// TIA Portal V17 export
// export: Created 2025-06-25T13:13:16.5727411Z, ExportSetting WithDefaults, DisplayName Totally Integrated Automation Portal, DisplayVersion V17 Update 8, DisplayName TIA Portal Openness, DisplayVersion V17 Update 8, DisplayName TIA Portal Version Control Interface, DisplayVersion V17, DisplayName STEP 7 Professional, DisplayVersion V17 Update 8, DisplayName STEP 7 Safety, DisplayVersion V17 Update 6, DisplayName WinCC Advanced, DisplayVersion V17 Update 8
FUNCTION "SaturationTemperature" : Real   // FC14, FBD
{ S7_Optimized_Access := 'TRUE' }
VERSION : 0.1
// stored: AutoNumber true, IsIECCheckEnabled false, SetENOAutomatically false, UDAEnableTagReadback false
   VAR_INPUT
      Pressure : Real;
   END_VAR
   VAR_IN_OUT
      Fluid : "FluidData-STRUCT";
   END_VAR
   VAR_TEMP
      MinPressure : Real;
   END_VAR
BEGIN

REGION Network 1
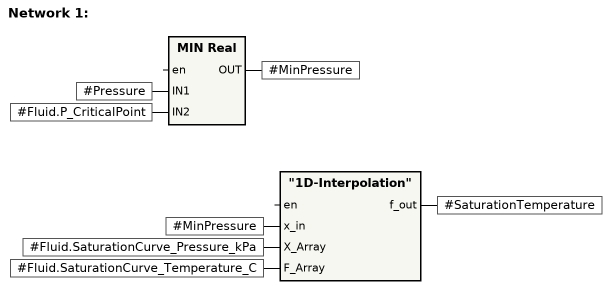
   #MinPressure := MIN(IN1 := #Pressure, IN2 := #Fluid.P_CriticalPoint);
   "1D-Interpolation"(x_in := #MinPressure,
                      X_Array := #Fluid.SaturationCurve_Pressure_kPa,
                      F_Array := #Fluid.SaturationCurve_Temperature_C,
                      f_out => #SaturationTemperature);
END_REGION
END_FUNCTION
